FUNCTION FC_AllStopped : BOOL
VAR_INPUT
	stStatus	:	ST_FSM_Status;
END_VAR
VAR
END_VAR

FC_AllStopped := (stStatus.stZ1.eStep = E_Z1_Step.Stop) AND
                 (stStatus.stZ2.eStep = E_Z2_Step.Stop) AND
                 (stStatus.stZ3.eStep = E_Z3_Step.Stop) AND	
                 (stStatus.stZ4.eStep = E_Z4_Step.Stop) AND
                 (stStatus.stZ5.eStep = E_Z5_Step.Stop) AND	
                 (stStatus.stZ6.eStep = E_Z6_Step.Stop);

END_FUNCTION

(* stored: Version 1.1.0.1
   POU FC_AllStopped: Id {a3e8e66f-6c96-0eff-012c-126d503c0501}, SpecialFunc None *)
